FUNCTION_BLOCK SET_CIRCLE_DATA (* Sets circle data to the proper format before sending to machine *)
  (* Standard: 61499-2 *)
  (* Version 1.0, 17-04-2012, GASR, Universidade do Estado de Santa Catarina *)
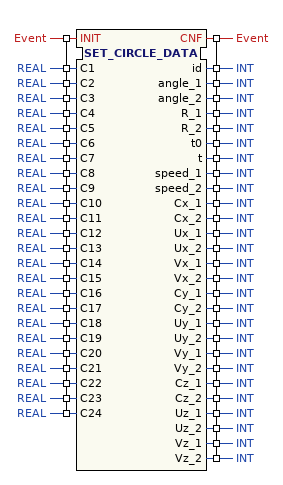
  EVENT_INPUT
    INIT WITH C1, C2, C3, C4, C5, C6, C7, C8, C9, C10, C11, C12, C13, C14, C15, C16, C17, C18, C19, C20, C21, C22, C23, C24;
  END_EVENT
  EVENT_OUTPUT
    CNF WITH id, angle_1, angle_2, R_1, R_2, t0, t, speed_1, speed_2, Cx_1, Cx_2, Ux_1, Ux_2, Vx_1, Vx_2, Cy_1, Cy_2, Uy_1, Uy_2, Vy_1, Vy_2, Cz_1, Cz_2, Uz_1, Uz_2, Vz_1, Vz_2;
  END_EVENT
  VAR_INPUT
    C1 : REAL; (* Coeficient 1 *)
    C2 : REAL; (* Coeficient 2 *)
    C3 : REAL; (* Coeficient 3 *)
    C4 : REAL; (* Coeficient 4 *)
    C5 : REAL; (* Coeficient 5 *)
    C6 : REAL; (* Coeficient 6 *)
    C7 : REAL; (* Coeficient 7 *)
    C8 : REAL; (* Coeficient 8 *)
    C9 : REAL; (* Coeficient 9 *)
    C10 : REAL; (* Coeficient 10 *)
    C11 : REAL; (* Coeficient 11 *)
    C12 : REAL; (* Coeficient 12 *)
    C13 : REAL; (* Coeficient 13 *)
    C14 : REAL; (* Coeficient 14 *)
    C15 : REAL; (* Coeficient 15 *)
    C16 : REAL; (* Coeficient 16 *)
    C17 : REAL; (* Coeficient 16 *)
    C18 : REAL; (* Coeficient 16 *)
    C19 : REAL; (* Coeficient 16 *)
    C20 : REAL; (* Coeficient 16 *)
    C21 : REAL; (* Coeficient 16 *)
    C22 : REAL; (* Coeficient 16 *)
    C23 : REAL; (* Coeficient 16 *)
    C24 : REAL; (* Coeficient 16 *)
  END_VAR
  VAR_OUTPUT
    id : INT;
    angle_1 : INT;
    angle_2 : INT;
    R_1 : INT;
    R_2 : INT;
    t0 : INT;
    t : INT;
    speed_1 : INT;
    speed_2 : INT;
    Cx_1 : INT;
    Cx_2 : INT;
    Ux_1 : INT;
    Ux_2 : INT;
    Vx_1 : INT;
    Vx_2 : INT;
    Cy_1 : INT;
    Cy_2 : INT;
    Uy_1 : INT;
    Uy_2 : INT;
    Vy_1 : INT;
    Vy_2 : INT;
    Cz_1 : INT;
    Cz_2 : INT;
    Uz_1 : INT;
    Uz_2 : INT;
    Vz_1 : INT;
    Vz_2 : INT;
  END_VAR
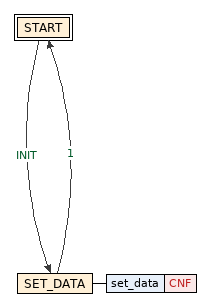
  EC_STATES
    START;
    SET_DATA : set_data -> CNF;
  END_STATES
  EC_TRANSITIONS
    START TO SET_DATA := INIT;
    SET_DATA TO START := 1;
  END_TRANSITIONS
  ALGORITHM set_data IN Lua:
function float_to_ints( n, precision )
	local n_1, n_2
	if( tonumber(n) >= 0 ) then
		n_1 = math.floor( n )
		n_2 = (n - n_1)*(10^precision)
		n_2 = math.floor( n_2 )
	else
		n_1 = math.ceil( n )
		n_2 = (n - n_1)*(10^precision)
		n_2 = math.ceil( n_2 )
	end
	return n_1, n_2
end

id = C1
angle_1, angle_2 = float_to_ints( C11, 3 )
R_1, R_2 = float_to_ints( C12, 3 )
t0 = C13
t = C14
print( 'Feed = ', C18 )
C18 = (C18/0.005)*60
print( 'Feed = ', C18 )
C18 = math.abs( C18 )
speed_1, speed_2 = float_to_ints( C18, 3 )
Cx_1, Cx_2 = float_to_ints( C2, 3 )
Ux_1, Ux_2 = float_to_ints( C5, 3 )
Vx_1, Vx_2 = float_to_ints( C8, 3 )
Cy_1, Cy_2 = float_to_ints( C3, 3 )
Uy_1, Uy_2 = float_to_ints( C6, 3 )
Vy_1, Vy_2 = float_to_ints( C9, 3 )
Cz_1, Cz_2 = float_to_ints( C4, 3 )
Uz_1, Uz_2 = float_to_ints( C7, 3 )
Vz_1, Vz_2 = float_to_ints( C10, 3 )
  END_ALGORITHM
END_FUNCTION_BLOCK
